// TIA Portal V20 export
TYPE "type_emRelations_em12_sequence"
// stored: Access Published, Namespace Unit1
   STRUCT
      stackNgBox : Struct
         jobs : "LAF_typeJobs";
         sequence : "LAF_typeSequence";
         selectJobStatus { S7_SetPoint := 'True'} : Array[0..10] of "LAF_typeJobStatus";
         "step" : "LER_typeStep";
         jobInterface : Struct
            loadJob2 : "LER_typeJobInterface";
            unloadJob3 : "LER_typeJobInterface";
         END_STRUCT;
         homeCheck : Struct
            partNoGet { ExternalWritable := 'False'} : Bool;
            partGet { ExternalWritable := 'False'} : Bool;
         END_STRUCT;
      END_STRUCT;
   END_STRUCT;
   // // stackNgBox."step".action1[101] : Step[101] : JOB[1] Condition
   // // stackNgBox."step".action1[110] : Step[110] : Clamp Z Up
   // // stackNgBox."step".action1[120] : Step[120] : Clamp Left, Right Open
   // // stackNgBox."step".action1[130] : Step[130] : Clamp Mover Open
   // // stackNgBox."step".action1[180] : Step[180] : Lift Down
   // // stackNgBox."step".action1[190] : Step[190] : JOB[1] Step End
   // // stackNgBox."step".action1[201] : Step[201] : JOB[2] Condition
   // // stackNgBox."step".action1[210] : Step[210] : Stack NG Box [Loading Request] => JR Unloading P&P
   // // stackNgBox."step".action1[220] : Step[220] : Clamp Mover Close
   // // stackNgBox."step".action1[230] : Step[230] : Clamp Left, Right Close
   // // stackNgBox."step".action1[231] : Step[231] : Stack NG Box [Loading Ready] => JR Unloading P&P
   // // stackNgBox."step".action1[290] : Step[290] : JOB[2] Step End
   // // stackNgBox."step".action1[301] : Step[301] : JOB[3] Condition
   // // stackNgBox."step".action1[310] : Step[310] : Clamp Z Down
   // // stackNgBox."step".action1[320] : Step[320] : Clamp Left, Right Open
   // // stackNgBox."step".action1[330] : Step[330] : Clamp Mover Open
   // // stackNgBox."step".action1[340] : Step[340] : Clamp Z Up
   // // stackNgBox."step".action1[390] : Step[390] : JOB[3] Step End
   // // stackNgBox."step".transition1[101] : Step[101] : JOB[1] Condition
   // // stackNgBox."step".transition1[110] : Step[110] : Clamp Z Up
   // // stackNgBox."step".transition1[120] : Step[120] : Clamp Left, Right Open
   // // stackNgBox."step".transition1[130] : Step[130] : Clamp Mover Open
   // // stackNgBox."step".transition1[180] : Step[180] : Lift Down
   // // stackNgBox."step".transition1[190] : Step[190] : JOB[1] Step End
   // // stackNgBox."step".transition1[201] : Step[201] : JOB[2] Condition
   // // stackNgBox."step".transition1[210] : Step[210] : Stack NG Box [Loading Request] => JR Unloading P&P
   // // stackNgBox."step".transition1[220] : Step[220] : Clamp Mover Close
   // // stackNgBox."step".transition1[230] : Step[230] : Clamp Left, Right Close
   // // stackNgBox."step".transition1[231] : Step[231] : Stack NG Box [Loading Ready] => JR Unloading P&P
   // // stackNgBox."step".transition1[290] : Step[290] : JOB[2] Step End
   // // stackNgBox."step".transition1[301] : Step[301] : JOB[3] Condition
   // // stackNgBox."step".transition1[310] : Step[310] : Clamp Z Down
   // // stackNgBox."step".transition1[320] : Step[320] : Clamp Left, Right Open
   // // stackNgBox."step".transition1[330] : Step[330] : Clamp Mover Open
   // // stackNgBox."step".transition1[340] : Step[340] : Clamp Z Up
   // // stackNgBox."step".transition1[390] : Step[390] : JOB[3] Step End
END_TYPE
